                    eStep := eCONNECTION_STATE_CONNECT_START;
                END_IF
            ELSE
                eStep := eCONNECTION_STATE_CLOSE_START;
            END_IF
        ELSIF bAccepted THEN
            eStep := eCONNECTION_STATE_DATAEXCHANGE;
        ELSE
            fbAcceptTimer( IN := FALSE, PT := T#0S );
        END_IF

    eCONNECTION_STATE_CONNECT_START:
        fbAccept( bExecute := FALSE );
        fbAccept( sSrvNetID := sSrvNetID,
                    hListener := hListener,
                    bExecute:= TRUE );
        eStep := eCONNECTION_STATE_CONNECT_WAIT;

    eCONNECTION_STATE_CONNECT_WAIT:
        fbAccept( bExecute := FALSE );
        IF NOT fbAccept.bBusy THEN
            IF NOT fbAccept.bError THEN
                IF fbAccept.bAccepted THEN
                    bAccepted := TRUE;
                    fbLog.Message( sMessage := 'Connection accepted!', hSocket := fbAccept.hSocket );
                END_IF
                eStep := eCONNECTION_STATE_IDLE;
            ELSE
                fbLog.Error( sMessage := 'FB_SocketAccept()', nErrId := fbAccept.nErrId );
                eStep := eCONNECTION_STATE_ERROR;
            END_IF
        END_IF

    eCONNECTION_STATE_DATAEXCHANGE:(* Data exchange state *)
        bDisconnect := NOT bEnable OR bDisconnect;(* User/internal disconnect requested? *)
        IF bDisconnect AND NOT bSndBusy AND NOT bRcvBusy THEN
            bDisconnect := FALSE;
            eStep := eCONNECTION_STATE_CLOSE_START;(* Disconnect *)
        ELSE

            (* Send tx data *)
            IF NOT bDisconnect AND NOT bSndBusy THEN
                //Test to fill output buffer to a higher degree if needed by trying to get several items from fbTx
                bGetMoreData:=TRUE;
                nTotalTxFrameReadLength:=0;
                WHILE bGetMoreData DO(* Success *)
                    fbTx.RemoveHead( bGet := ADR(bTxFrame[nTotalTxFrameReadLength]), nReadCount=>nTxFrameReadLength,nReadBufferSize:=(SIZEOF(bTxFrame)-nTotalTxFrameReadLength));(* Remove oldest string entry s*)
                    bGetMoreData:= fbTx.bOk;
                    IF bGetMoreData THEN
                        nTotalTxFrameReadLength:=nTotalTxFrameReadLength+nTxFrameReadLength; //only inrease counter if successfull
                    END_IF;
                END_WHILE
                IF nTotalTxFrameReadLength>0 THEN
                    sTxBuffer:=ADR(bTxFrame); //Just to se the data in string format
                    fbSend( bExecute := FALSE );
                    fbSend( sSrvNetID := sSrvNetID,
                            hSocket := fbAccept.hSocket,
                            pSrc    := ADR( bTxFrame ),
                            cbLen   := DINT_TO_UINT(nTotalTxFrameReadLength),//INT_TO_UDINT(LEN( sTxFrame )) (*+ 1*),(* String length inclusive the zero delimiter *) (*Commented away because to much was sent to host (one '.' to much) *)
                            bExecute:= TRUE );
                    bSndBusy := TRUE;
                END_IF

                (*fbTx.RemoveHead( bGet := ADR(bTxFrame), nReadCount=>nTxFrameReadLength,nReadBufferSize:=SIZEOF(bTxFrame) );(* Remove oldest string entry s*)
                IF fbTx.bOk THEN(* Success *)
                    sTxBuffer:=ADR(bTxFrame); //Just to se the data in string format
                    fbSend( bExecute := FALSE );
                    fbSend( sSrvNetID := sSrvNetID,
                            hSocket := fbAccept.hSocket,
                            pSrc    := ADR( bTxFrame ),
                            cbLen   := nTxFrameReadLength,//INT_TO_UDINT(LEN( sTxFrame )) (*+ 1*),(* String length inclusive the zero delimiter *) (*Commented away because to much was sent to host (one '.' to much) *)
                            bExecute:= TRUE );
                    bSndBusy := TRUE;
                END_IF
                *)
            ELSE
                fbSend( bExecute := FALSE );
                IF NOT fbSend.bBusy THEN
                    bSndBusy := FALSE;
                    IF fbSend.bError THEN
                        fbLog.Error( sMessage := 'FB_SocketSend()', nErrId := fbSend.nErrId );
                        bDisconnect := TRUE;(* Set flag *)
                    END_IF
                END_IF
            END_IF


            (* Get rx data *)
            IF NOT bDisconnect AND NOT bRcvBusy THEN
                fbPollTimer( IN := TRUE );
                IF fbPollTimer.Q THEN
                    fbPollTimer( IN := FALSE, PT := PLCPRJ_RECEIVE_POLLING_TIME );
                    fbReceive( bExecute := FALSE );
                    fbReceive(  sSrvNetID := sSrvNetID,
                                hSocket := fbAccept.hSocket,
                                pDest   := ADR( rxBuffer ) + cbReceived,
                                cbLen   := SIZEOF( rxBuffer ) - cbReceived,
                                bExecute:= TRUE );
                    bRcvBusy := TRUE;
                END_IF
            ELSE
                fbReceive( bExecute := FALSE );
                IF NOT fbReceive.bBusy THEN
                    bRcvBusy := FALSE;
                    IF NOT fbReceive.bError THEN
                        IF (fbReceive.nRecBytes > 0) THEN(* Bytes received *)

                            fbPollTimer( IN := FALSE, PT := T#0S ); (* Bytes received => increase the read (polling) speed *)
                            fbRequestTimer( IN := FALSE );(* Bytes received => disable timeout check *)
                            cbReceived  := cbReceived + fbReceive.nRecBytes;(* Calculate the number of received data bytes *)

                            //Move to input queue
                            IF cbReceived>0 AND cbReceived<PLCPRJ_BUFFER_SIZE-1 AND cbReceived< fbRx.cbFree THEN
                                fbRx.AddTail( bPut := ADR(rxBuffer),nWriteCount:=UDINT_TO_INT(cbReceived));(* Put received message to the rx fifo *)
                                cbReceived:=0;
                                IF NOT fbRx.bOk THEN
                                    fbLog.Error( sMessage := 'FB_FrameFifo(receiver)', nErrID := PLCPRJ_ERROR_RECFIFO_OVERFLOW );
                                    bDisconnect := TRUE;(* Set flag *)
                                    RETURN;
                                END_IF

                            END_IF

                            //REPEAT

                                (* Search for string end delimiter *)
                            //  nLenOfString := 0;(* Reset string length *)
                            //  bEndOfString := FALSE;
                            //  REPEAT
                            //      IF rxBuffer[nLenOfString] = 10 THEN(* String end delimiter found Line feed *)
                            //          bEndOfString := TRUE;
                            //      END_IF
                            //      nLenOfString := nLenOfString + 1;
                            //  UNTIL bEndOfString OR (nLenOfString >= cbReceived)
                            //  END_REPEAT

                            //  IF bEndOfString THEN
                            //      MEMSET( ADR( bRxFrame ), 0, SIZEOF( bRxFrame ) );
                            //      MEMCPY(  ADR( bRxFrame ), ADR( rxBuffer ), MIN( SIZEOF(bRxFrame), nLenOfString ) );(* Copy the received string to the output variable (inclusive the end delimiter) *)
                            //      MEMMOVE( ADR( rxBuffer ), ADR( rxBuffer[nLenOfString] ), cbReceived - nLenOfString  );(* Move the reamaining data bytes *)
                            //      cbReceived := cbReceived - nLenOfString;(* Recalculate the reamaining data byte length *)

                            //      fbRx.AddTail( bPut := bRxFrame );(* Put received message to the rx fifo *)
                            //      IF NOT fbRx.bOk THEN
                            //          fbLog.Error( sMessage := 'FB_FrameFifo(receiver)', nErrID := PLCPRJ_ERROR_RECFIFO_OVERFLOW );
                            //          bDisconnect := TRUE;(* Set flag *)
                            //          RETURN;
                            //      END_IF
                            //  END_IF

                            //UNTIL NOT bEndOfString OR (cbReceived = 0)
                            //END_REPEAT

                        ELSE(* No bytes received *)
                            fbRequestTimer( IN := TRUE, PT := PLCPRJ_RECEIVE_TIMEOUT );(* No bytes received => enable timeout check *)
                            IF fbRequestTimer.Q THEN (* Timeout error*)
                            //  fbRequestTimer( IN := FALSE );
                            //  fbLog.Error( sMessage := 'FB_SocketReceive()', nErrID := PLCPRJ_ERROR_RECEIVE_TIMEOUT );
                            //  bDisconnect := TRUE;(* Set flag *)
                            END_IF
                        END_IF

                    ELSE(* Receive error *)
                        fbLog.Error( sMessage := 'FB_SocketReceive()', nErrId := fbReceive.nErrId );
                        bDisconnect := TRUE;(* Set flag *)
                    END_IF
                END_IF(* IF NOT fbReceive.bBusy THEN *)

            END_IF(* IF NOT bDisconnect AND NOT bRcvBusy THEN *)

        END_IF(* IF bDisconnect AND NOT bSndBusy AND NOT bRcvBusy THEN *)



    eCONNECTION_STATE_CLOSE_START:
        fbLog.Message( sMessage := 'Closing connection!', hSocket := fbAccept.hSocket );
        fbClose( bExecute := FALSE );
        fbClose( sSrvNetID := sSrvNetID, hSocket:= fbAccept.hSocket, bExecute:= TRUE );
        eStep := eCONNECTION_STATE_CLOSE_WAIT;

    eCONNECTION_STATE_CLOSE_WAIT:
        fbClose( bExecute := FALSE );
        IF NOT fbClose.bBusy THEN
            bAccepted := FALSE;
            IF NOT fbClose.bError THEN
                eStep := eCONNECTION_STATE_IDLE;
            ELSE
                fbLog.Error( sMessage := 'FB_SocketClose(accepted)', nErrId := fbClose.nErrId );
                eStep := eCONNECTION_STATE_ERROR;
            END_IF
        END_IF

    eCONNECTION_STATE_ERROR:
        IF bAccepted THEN
            eStep := eCONNECTION_STATE_CLOSE_START;
        ELSE
            eStep := eCONNECTION_STATE_IDLE;
        END_IF

END_CASE

END_FUNCTION_BLOCK

// ---- POUs/Helper POUs/CheckBounds.TcPOU
FUNCTION CheckBounds : DINT
VAR_INPUT
        index, lower, upper : DINT;
END_VAR
VAR
END_VAR

IF index<lower THEN
        CheckBounds := lower;
ELSIF index>upper THEN
        CheckBounds := upper;
ELSE
        CheckBounds := index;
END_IF

END_FUNCTION

// ---- POUs/README.TcPOU
PROGRAM README
VAR
    sVersion: STRING:='0.9.0';
END_VAR

(*

The EpicsComModule is used to communicate between EPICS and a TwinCAT 3 PLC (Beckhoff). The communication between epics and this module is based on TCP/IP (Stream device is used on the EPICS-side). Internal communication between this module and other modules (other plc-modules, motion-module, or I/O) are based on ADS communication.
The EpicsComModule currently utilizes the Beckhoff TCP/IP server framework. Therefore the TCP/IP server software needs to be installed on the controller to be used. A licence for the TCP/IP server must be activated if it should run more than 7-days continiuosly (like all TwinCat licenses).
Note: No lcence is needed to test for 7 days (test period will autamaticcaly be renewed to 7 more days each time the project is downloaded)

Quick start guide:
0: Read the manual
1: Add the EpicsComModule to your project (easiest way is to use add existing item (right click on PLC in treeview)). Or use git
2: Compile and download:
3: Configure records in EPICS (Using steram device) to output strings in the following format:
    Read a varaible: "Main.iCounter?;
"
    Write a variable: "Main.iCounter=10;
"
The default internal ADS adress is 851 which corresponds to the first PLC-module (Main.iCounter in PLC module 851 will be accessed). For accessing other ADS-modules please refer to documentation.

Most native types and arrays of native types are supported (also some structs).


******* Other functionallity **********

****Options (options are defined by an ending '/'):
"ADSPORT=xxx/Command;" Will apply a ADS-port to an command. This ADS port will only be used for the command stated after the option. The default ADS-port will be unchanged
example:
    "ADSPORT=852/Main.iCounter?;"   Will access Main.iCounter on ADS port 852.

****Commands (Commands are identified by an '.' located at the first byte in the command string):
".THIS.XXXXXX;" Will allow access to variables in the current communication object. (since the client don't know which to connection object in the array it's connected to )
example:
".THIS.stSettings.nADSPORT=852;" will change the default ADS-port to 852.  .THIS will simply replace  the path to the communication object with the correct connection index (x):
".THIS.stSettings.nADSPORT=852;" = "Main.fbServer.aApplications[x].stSettings.nADSPORT=852;"
example 2:
".THIS.stSettings.nConnectionIndex?;" will retrun the connection index for the current connection.


".ADR.IDXGRP,IDXOFF,size,adst_type;". The ADR command allows reading and writing to variables with absoulte adress
example: Access softlimits of axis 1 in motion (NC). Adresses can be find in documentation on by hovering over the parameter in NC (tool tip) or by right clicking on the parameter of intrest and choosing properties. NC has ADSPort 501
Writing: "ADSPORT=501/.ADR.16#5001,16#D,8,5=-100;"
Reading: "ADSPORT=501/.ADR.16#5001,16#D,8,5?;"
Note: Axis 2 can be accessed in the same way by increasing the IDXGRP to 5002  (axis 3=> 5003)

example 2: Reading the absoute adress of an variable with symbolic adress

"ADSPORT=852/.ADR.Main.sVersion?; Will return the absolute adress of the variable Main.sVersion at ADS-port 852.

*)

END_PROGRAM

// ---- POUs/Static Command support/FB_GetStaticADR.TcPOU
FUNCTION_BLOCK FB_GetStaticADR
VAR
    sVersion: STRING:='0.9.0';
END_VAR
VAR_INPUT
    bEnable:BOOL:=FALSE;
    nCommadStartIndex:INT:=0;
    nCommandEndIndex:INT:=0;
END_VAR
VAR
    psCommandBufferString: POINTER TO STRING; //string to point into byte buffer
    nQuestionSign: INT;
END_VAR

VAR_IN_OUT
    byteCommandBuffer   :   ARRAY[0..PLCPRJ_BUFFER_SIZE] OF BYTE;//ADS input buffer
    nBytesInCommandBuffer:DINT:=0;
    nIndexEndOfCommand:DINT:=0;
END_VAR

VAR_OUTPUT
    nErrorId: UDINT;
    bError:BOOL:=FALSE;
    sVariableName:STRING(255);
    sSubErrorString: STRING;
END_VAR

//Static command/option 1: Check if ADR option
(*IF bEnable THEN
    bError:=FALSE;
    nErrorId:=0;
    sSubErrorString:='';
    sVariableName:='';
    psCommandBufferString:=ADR(byteCommandBuffer);
    nQuestionSign:=len(STR:=EPICS_STATIC_COMMAND_ABS_ADRESS);
    IF  byteCommandBuffer[len(STR:=EPICS_STATIC_COMMAND_ABS_ADRESS)]=EPICS_ASCII_QUESTIONMARK AND nQuestionSign>0 THEN
        sVariableName:=right(str:=left(str:=PSTRING_TO_STRING(psCommandBufferString),size:=nCommandEndIndex-1),SIZE:=(nCommandEndIndex-1)-nQuestionSign-1);
        IF NOT F_RemoveBytesFromBuffer_V1_00(nRemoveBytes:= nCommandEndIndex,byteCommandBuffer:=byteCommandBuffer,nBytesInCommandBuffer:=nBytesInCommandBuffer,nIndexEndOfCommand:=nIndexEndOfCommand) THEN
            bError:=TRUE;
            nErrorId:=312;
            sSubErrorString:='State 3: Failed to clear buffer (ADR).';
        END_IF
    ELSE
        nErrorId:=313;
        bError:=TRUE;
        sSubErrorString:='State 3: Failed to parse ADR set command.';
    END_IF
END_IF*)

END_FUNCTION_BLOCK

// ---- POUs/Static Command support/FB_ParseStaticCommand.TcPOU
FUNCTION_BLOCK FB_ParseStaticCommand
VAR
    sVersion: STRING:='0.9.0';
END_VAR
VAR
    psCommandBufferString: POINTER TO STRING; //string to point into byte buffer
    nEqualSign: INT;
    nQuestionMark: INT;
END_VAR

VAR_IN_OUT
    byteCommandBuffer   :   ARRAY[0..PLCPRJ_BUFFER_SIZE] OF BYTE;//ADS input buffer
    nBytesInCommandBuffer:DINT:=0;
    nIndexEndOfCommand:DINT:=0;
END_VAR

VAR_OUTPUT
    nErrorId: UDINT;
    bError:BOOL:=FALSE;
    sSubErrorString: STRING;
    sStaticCommand:STRING;
    sStaticValue:STRING;
    bReadCommand:BOOL:=FALSE;
    bWriteCommand:BOOL:=FALSE;
END_VAR

//Parse static command
nErrorId:=0;
bError:=FALSE;
sStaticCommand:='';
sStaticValue:='';
bReadCommand:=FALSE;
bWriteCommand:=FALSE;
psCommandBufferString:=ADR(byteCommandBuffer);

nEqualSign:=find(STR1:=PSTRING_TO_STRING(psCommandBufferString),STR2:=EPICS_WRITE_CMD);
IF nEqualSign>0 AND nEqualSign<=nIndexEndOfCommand THEN
    bWriteCommand:=TRUE;
    //Command
    memcpy(destAddr:=ADR(sStaticCommand[0]),srcAddr:=ADR(byteCommandBuffer[0]),n:=nEqualSign-1);
    memset(destAddr :=ADR(sStaticCommand[nEqualSign-1]),fillByte:=0,n:=1);              //Terminate string
    //Value
    memcpy(destAddr:=ADR(sStaticValue[0]),srcAddr:=ADR(byteCommandBuffer[nEqualSign]),n:=nIndexEndOfCommand-nEqualSign-1);
    memset(destAddr :=ADR(sStaticValue[nIndexEndOfCommand-nEqualSign-1]),fillByte:=0,n:=1); //Terminate string
    IF NOT F_RemoveBytesFromBuffer_V1_00(nRemoveBytes:= nIndexEndOfCommand,byteCommandBuffer:=byteCommandBuffer,nBytesInCommandBuffer:=nBytesInCommandBuffer,nIndexEndOfCommand:=nIndexEndOfCommand) THEN
        bError:=TRUE;
        nErrorId:=301;
        sSubErrorString:='State 3: Failed to clear buffer (Parse static command write).';
    END_IF
ELSE
    nQuestionMark:=find(STR1:=PSTRING_TO_STRING(psCommandBufferString),STR2:=EPICS_READ_CMD);
    IF nQuestionMark>0 AND nQuestionMark<=nIndexEndOfCommand THEN
        bReadCommand:=TRUE;
        //Command
        memcpy(destAddr:=ADR(sStaticCommand[0]),srcAddr:=ADR(byteCommandBuffer[0]),n:=nQuestionMark-1);
        memset(destAddr :=ADR(sStaticCommand[nQuestionMark-1]),fillByte:=0,n:=1);               //Terminate string

        //Clean buffer
        IF NOT F_RemoveBytesFromBuffer_V1_00(nRemoveBytes:= nIndexEndOfCommand,byteCommandBuffer:=byteCommandBuffer,nBytesInCommandBuffer:=nBytesInCommandBuffer,nIndexEndOfCommand:=nIndexEndOfCommand) THEN
            bError:=TRUE;
            nErrorId:=302;
            sSubErrorString:='State 3: Failed to clear buffer (Parse static command read).';
        END_IF
    END_IF
END_IF

IF NOT (bReadCommand OR  bWriteCommand) THEN
    bError:=TRUE;
    nErrorId:=303;
    sSubErrorString:='State 3: Parsing of static command failed.';
END_IF

END_FUNCTION_BLOCK

// ---- POUs/Static Command support/FB_SetStaticADSPort.TcPOU
FUNCTION_BLOCK FB_SetStaticADSPort
VAR
    sVersion: STRING:='0.9.0';
END_VAR
VAR_INPUT
    bEnable:BOOL:=FALSE;
    nCommadStartIndex:INT:=0;
    nCommandEndIndex:INT:=0;
END_VAR
VAR
    psCommandBufferString: POINTER TO STRING; //string to point into byte buffer
    bInStaticSection: BOOL;
    sTemp: STRING;
    nEqualSign: INT;
END_VAR

VAR_IN_OUT
    byteCommandBuffer   :   ARRAY[0..PLCPRJ_BUFFER_SIZE] OF BYTE;//ADS input buffer
    nBytesInCommandBuffer:DINT:=0;
    nIndexEndOfCommand:DINT:=0;
END_VAR

VAR_OUTPUT
    nErrorId: UDINT;
    bError:BOOL:=FALSE;
    nADSPort: UINT:=0;
    sSubErrorString: STRING;
END_VAR

//Static command/option 1: Check if ADSPORT option
IF bEnable THEN
    psCommandBufferString:=ADR(byteCommandBuffer);
    nEqualSign:=find(STR1:=PSTRING_TO_STRING(psCommandBufferString),STR2:=EPICS_WRITE_CMD);
    sTemp:=right(str:=left(str:=PSTRING_TO_STRING(psCommandBufferString),size:=nCommandEndIndex-1),SIZE:=(nCommandEndIndex-1)-nEqualSign);
    nADSPort:=STRING_TO_UINT(sTemp);
    IF nADSPort<1 OR nADSPort>20000 THEN
        nErrorId:=301;
        bError:=TRUE;
        sSubErrorString:='State 3: ADSPORT out of range.';
    //  nADSPort:=EPICS_ADS_PORT; //Set to default
    END_IF
    //Remove ADS command from buffer
    IF NOT F_RemoveBytesFromBuffer_V1_00(nRemoveBytes:= nCommandEndIndex,byteCommandBuffer:=byteCommandBuffer,nBytesInCommandBuffer:=nBytesInCommandBuffer,nIndexEndOfCommand:=nIndexEndOfCommand) THEN
            bError:=TRUE;
            nErrorId:=302;
            sSubErrorString:='State 3: Failed to clear buffer (ADSPORT)).';
    END_IF
END_IF

END_FUNCTION_BLOCK

// ---- POUs/Static Command support/FB_SetStaticADR.TcPOU
FUNCTION_BLOCK FB_SetStaticADR
VAR
    sVersion: STRING:='0.9.0';
END_VAR
VAR_INPUT
    bEnable:BOOL:=FALSE;
    nCommadStartIndex:INT:=0;
    nCommandEndIndex:INT:=0;
END_VAR
VAR
    psCommandBufferString: POINTER TO STRING; //string to point into byte buffer
    bInStaticSection: BOOL;
    sTemp: STRING;
    nEqualSign: INT;
    nComma:INT:=0;
    stemp1: STRING(255);
    sTemp2: STRING(255);
    sTemp3: STRING(255);
    sTemp4: STRING(255);
    sVal:STRING;
    nQuestionSign: INT;
    nRemove: INT;
END_VAR

VAR_IN_OUT
    byteCommandBuffer   :   ARRAY[0..PLCPRJ_BUFFER_SIZE] OF BYTE;//ADS input buffer
    nBytesInCommandBuffer:DINT:=0;
    nIndexEndOfCommand:DINT:=0;
END_VAR

VAR_OUTPUT
    nErrorId: UDINT;
    bError:BOOL:=FALSE;
    stSymInfo:SYMINFOSTRUCT;
    sSubErrorString: STRING;
END_VAR

//Should look like "ADR=idxgrp,idxoff,size,type/"   => ADR=1,2,3,4/
(*
Type:
ADST_BIT             = 33 (&H21)
ADST_INT8            = 16 (&H10)
ADST_INT16           = 2
ADST_INT32           = 3
ADST_INT64           = 20 (&H14)
ADST_UINT8           = 17 (&H11)
ADST_UINT16          = 18 (&H12)
ADST_UINT32          = 19 (&H13)
ADST_UINT64          = 21 (&H15)
ADST_REAL32          = 4
ADST_REAL64          = 5
ADST_REAL80          = 32 (&H20)
ADST_BIGTYPE         = 65 (&H41)
ADST_VOID            = 0
*)

//Static command/option 1: Check if ADR option
IF bEnable THEN
    bError:=TRUE;
    nErrorId:=0;
    sSubErrorString:='';
    stSymInfo.adsDataType:=0;
    stSymInfo.byteSize:=0;
    stSymInfo.idxGroup:=0;
    stSymInfo.idxOffset:=0;
    nRemove:=0;
    psCommandBufferString:=ADR(byteCommandBuffer);
    nEqualSign:=find(STR1:=PSTRING_TO_STRING(psCommandBufferString),STR2:=EPICS_WRITE_CMD);
    sTemp:=right(str:=left(str:=PSTRING_TO_STRING(psCommandBufferString),size:=nCommandEndIndex-1),SIZE:=(nCommandEndIndex)-nEqualSign-1);
    nComma:=find(STR1:=sTemp,STR2:=EPICS_ARRAY_DELIMITER);
    IF  nComma>0 THEN
        sVal:=left(STR:=sTemp,size:=nComma);
        stSymInfo.idxGroup:=STRING_TO_UDINT(sVal);
        sTemp1:=right(STR:=sTemp,size:=len(sTemp)-nComma);
        nRemove:=nRemove+nComma+1;
        nComma:=find(STR1:=sTemp1,STR2:=EPICS_ARRAY_DELIMITER);
        IF  nComma>0 THEN
            sVal:=left(STR:=sTemp1,size:=nComma);
            stSymInfo.idxOffset:=STRING_TO_UDINT(sVal);
            sTemp2:=right(STR:=sTemp1,size:=len(sTemp1)-nComma);
            nRemove:=nRemove+nComma+1;
            nComma:=find(STR1:=sTemp2,STR2:=EPICS_ARRAY_DELIMITER); //last
            IF  nComma>0 THEN
                sVal:=left(STR:=sTemp2,size:=nComma);
                stSymInfo.byteSize:=STRING_TO_UDINT(sVal);
                sTemp3:=right(STR:=sTemp2,size:=len(sTemp2)-nComma);
                nRemove:=nRemove+nComma+1;
                nComma:=len(sTemp3);
                IF nComma>0 AND find(str1:=stemp3,str2:=EPICS_COMMAND_OPTION_DELIMITER)=0 THEN
                    stSymInfo.adsDataType:=STRING_TO_INT(sTemp3);
                    nRemove:=nRemove+nComma+1;
                    bError:=FALSE;
                END_IF
            END_IF
        END_IF
    END_IF

    IF bError THEN
        nErrorId:=310;
        bError:=TRUE;
        sSubErrorString:='State 3: Failed to parse ADR command.';
        // try to clean buffers
        F_RemoveBytesFromBuffer_V1_00(nRemoveBytes:= nRemove,byteCommandBuffer:=byteCommandBuffer,nBytesInCommandBuffer:=nBytesInCommandBuffer,nIndexEndOfCommand:=nIndexEndOfCommand);
    ELSE
        IF NOT F_RemoveBytesFromBuffer_V1_00(nRemoveBytes:= nCommandEndIndex,byteCommandBuffer:=byteCommandBuffer,nBytesInCommandBuffer:=nBytesInCommandBuffer,nIndexEndOfCommand:=nIndexEndOfCommand) THEN
            bError:=TRUE;
            nErrorId:=311;
            sSubErrorString:='State 3: Failed to clear buffer (ADR).';
        END_IF
    END_IF
END_IF

END_FUNCTION_BLOCK
